// TIA Portal project "EJERCICIO ANALOGIA" (V11)

(* hardware
DEVICE "S7300/ET200 station_1"  SIMATIC 300-Station
   slot 0: "Perfil soporte_0"  Rail  6ES7 390-1***0-0AA0
   slot 2: "PLC_1"  CPU 313C-2 DP  6ES7 313-6CF03-0AB0  V2.6
      slot 0: "Interfaz MPI_1"  MPI
      slot 1: "Interfaz DP_1"  DP
      slot 2: "DI16/DO16_1"  DI16/DO16
      slot 4: "Contaje_1"  Counter
*)

// ===== PLC "PLC_1"  CPU 313C-2 DP =====

VAR_GLOBAL   // PLC tag table "Tabla de variables estándar"
   "Tag_1" AT %E0.0 : Bool;
   "SEÑAL ANALOGICA" AT %MD0 : Real;
   "SALIDA ESCALADO" AT %MD4 : Real;
   "PROPORCIONAL" AT %MD8 : Real;
   "DERIVATIVO" AT %MD12 : Real;
   "INTEGRAL" AT %MD16 : Real;
   "PID" AT %MD20 : Real;
   "BP" AT %MD24 : Real;
   "D" AT %MD28 : Real;
   "I" AT %MD32 : Real;
   "SP" AT %MD36 : Real;
   "valor desescaldo pid" AT %MD40 : Real;
   "porcrntaje apertura valvula" AT %MD44 : Real;
END_VAR

DATA_BLOCK "ESCALADOX_DB"   // DB1
{ S7_Optimized_Access := 'FALSE' }
VERSION : 0.1
// stored: InstanceOfName ESCALADOX
"ESCALADOX"
BEGIN
END_DATA_BLOCK

DATA_BLOCK "DESESCALADO_DB"   // DB2
{ S7_Optimized_Access := 'FALSE' }
VERSION : 0.1
// stored: InstanceOfName DESESCALADO
"DESESCALADO"
BEGIN
END_DATA_BLOCK

DATA_BLOCK "CONTROL PID_DB"   // DB3
{ S7_Optimized_Access := 'FALSE' }
VERSION : 0.1
// stored: InstanceOfName CONTROL PID
"CONTROL PID"
BEGIN
END_DATA_BLOCK

DATA_BLOCK "ESCALADOX_DB_1"   // DB8
{ S7_Optimized_Access := 'FALSE' }
VERSION : 0.1
// stored: InstanceOfName ESCALADOX
"ESCALADOX"
BEGIN
END_DATA_BLOCK

FUNCTION_BLOCK "CONTROL PID"   // FB1, SCL
{ S7_Optimized_Access := 'FALSE' }
VERSION : 0.1
   VAR_INPUT
      SP : Real;
      PV : Real;
      PB : Real;
      D : Real;
      I : Real;
   END_VAR
   VAR_OUTPUT
      "POULT PRO" : Real;
      "POULT DERI" : Real;
      "POULT INTE" : Real;
      "POULT PID PRO" : Real;
   END_VAR
   VAR
      M0 : Bool;
      M1 : Bool;
      T0 : Bool;
      T1 : Bool;
      T2 : Bool;
      T3 : Bool;
      "VISUALIZAR 0" : Time;
      "VISUALIZAR 1" : Time;
      "VISUALIZAR 2" : Time;
      "VISUALIZAR 3" : Time;
      "valor PB" : Real;
      "PB 75 %" : Real;
      "error der inicial" : Real;
      "error int inicial" : Real;
      "error der final" : Real;
      "error int final" : Real;
      ERROR : Real;
      Kp : Real;
      poult : Real;
      Kd : Real;
      "poult der" : Real;
      "diferencia error" : Real;
      Ki : Real;
      "poult int" : Real;
      "incremento error" : Real;
      "aux error integ" : Real;
      "poult pid" : Real;
      Nº100 : Real := 100.0;
      Nº : Real := 0.25;
   END_VAR
BEGIN
END_FUNCTION_BLOCK

FUNCTION_BLOCK "ESCALADOX"   // FB2, SCL
{ S7_Optimized_Access := 'FALSE' }
VERSION : 0.1
   VAR_INPUT
      Y2 : Real;
      Y1 : Real;
      X2 : Real;
      X1 : Real;
      CALCULAR : Bool;
      x : Real;
   END_VAR
   VAR_OUTPUT
      resultado : Real;
   END_VAR
   VAR
      Y : Real;
      "PENDIENTE (m)" : Real;
      "PUNTOCORTE (n)" : Real;
   END_VAR
BEGIN

     #"PENDIENTE (m)" :=  (#Y2 - (#Y1) ) / ( #X2 -#X1   )  ;
     #"PUNTOCORTE (n)" := #Y2  -  #"PENDIENTE (m)" * #X2   ;
     #resultado:= ( #"PENDIENTE (m)" * #x ) + #"PUNTOCORTE (n)";
END_FUNCTION_BLOCK

FUNCTION_BLOCK "DESESCALADO"   // FB3, SCL
{ S7_Optimized_Access := 'FALSE' }
VERSION : 0.1
   VAR_INPUT
      Y2 : Real;
      Y1 : Real;
      X2 : Real;
      X1 : Real;
      "y  valor a desescalar" : Real;
   END_VAR
   VAR_OUTPUT
      "X valor desescalado" : Real;
   END_VAR
   VAR
      "PENDIENTE ( m )" : Real;
      "PUNTO DE CORTE (n )" : Real;
   END_VAR
BEGIN

    #"PENDIENTE ( m )" :=  (#Y2 - (#Y1) ) / ( #X2 -#X1   )  ;
    #"PUNTO DE CORTE (n )" := #Y2  - #"PENDIENTE ( m )" * #X2   ;
    #"X valor desescalado" :=(#"y  valor a desescalar" / #"PENDIENTE ( m )" ) - #"PUNTO DE CORTE (n )" ;
END_FUNCTION_BLOCK

ORGANIZATION_BLOCK "Main"   // OB1, LAD
TITLE = "Main Program Sweep (Cycle)"
{ S7_Optimized_Access := 'FALSE' }
VERSION : 0.1
   VAR_TEMP
      OB1_EV_CLASS : Byte;   // Bits 0-3 = 1 (Coming event), Bits 4-7 = 1 (Event class 1)
      OB1_SCAN_1 : Byte;   // 1 (Cold restart scan 1 of OB 1), 3 (Scan 2-n of OB 1)
      OB1_PRIORITY : Byte;   // Priority of OB Execution
      OB1_OB_NUMBR : Byte;   // 1 (Organization block 1, OB1)
      OB1_RESERVED_1 : Byte;   // Reserved for system
      OB1_RESERVED_2 : Byte;   // Reserved for system
      OB1_PREV_CYCLE : Int;   // Cycle time of previous OB1 scan (milliseconds)
      OB1_MIN_CYCLE : Int;   // Minimum cycle time of OB1 (milliseconds)
      OB1_MAX_CYCLE : Int;   // Maximum cycle time of OB1 (milliseconds)
      OB1_DATE_TIME : Date_And_Time;   // Date and time OB1 started
   END_VAR
BEGIN

REGION Network 1
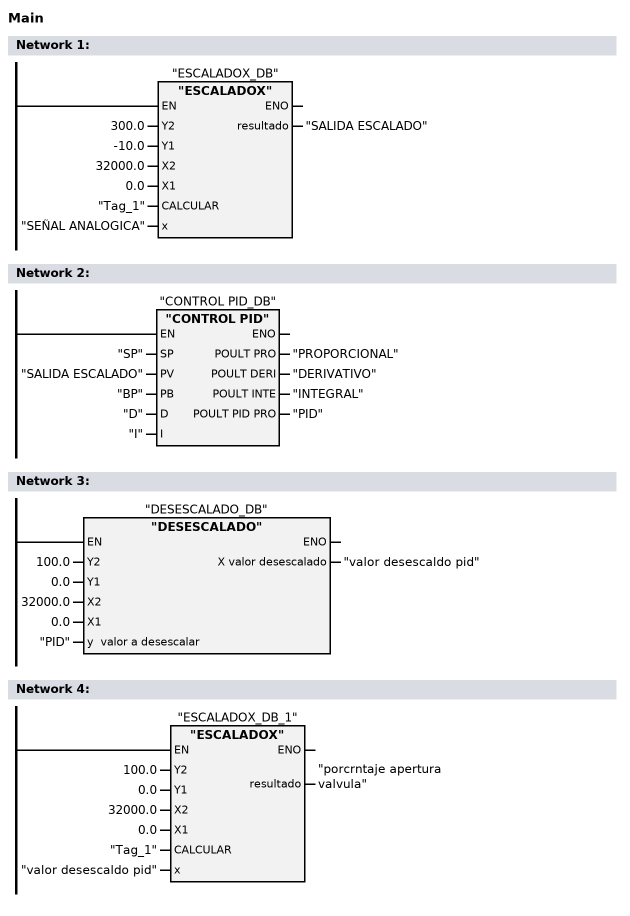
   RUNG wire#powerrail
      "ESCALADOX_DB"(Y2 := 300.0, Y1 := -10.0, X2 := 32000.0, X1 := 0.0, CALCULAR := "Tag_1", x := "SEÑAL ANALOGICA", resultado => "SALIDA ESCALADO")
   END_RUNG
   // the same network as SCL:
   "ESCALADOX_DB"(Y2 := 300.0,   // "ESCALADOX"
                  Y1 := -10.0,
                  X2 := 32000.0,
                  X1 := 0.0,
                  CALCULAR := "Tag_1",
                  x := "SEÑAL ANALOGICA",
                  resultado => "SALIDA ESCALADO");
END_REGION

REGION Network 2
   RUNG wire#powerrail
      "CONTROL PID_DB"(SP := "SP", PV := "SALIDA ESCALADO", PB := "BP", D := "D", I := "I", "POULT PRO" => "PROPORCIONAL", "POULT DERI" => "DERIVATIVO", "POULT INTE" => "INTEGRAL", "POULT PID PRO" => "PID")
   END_RUNG
   // the same network as SCL:
   "CONTROL PID_DB"(SP := "SP",   // "CONTROL PID"
                    PV := "SALIDA ESCALADO",
                    PB := "BP",
                    D := "D",
                    I := "I",
                    "POULT PRO" => "PROPORCIONAL",
                    "POULT DERI" => "DERIVATIVO",
                    "POULT INTE" => "INTEGRAL",
                    "POULT PID PRO" => "PID");
END_REGION

REGION Network 3
   RUNG wire#powerrail
      "DESESCALADO_DB"(Y2 := 100.0, Y1 := 0.0, X2 := 32000.0, X1 := 0.0, "y  valor a desescalar" := "PID", "X valor desescalado" => "valor desescaldo pid")
   END_RUNG
   // the same network as SCL:
   "DESESCALADO_DB"(Y2 := 100.0,   // "DESESCALADO"
                    Y1 := 0.0,
                    X2 := 32000.0,
                    X1 := 0.0,
                    "y  valor a desescalar" := "PID",
                    "X valor desescalado" => "valor desescaldo pid");
END_REGION

REGION Network 4
   RUNG wire#powerrail
      "ESCALADOX_DB_1"(Y2 := 100.0, Y1 := 0.0, X2 := 32000.0, X1 := 0.0, CALCULAR := "Tag_1", x := "valor desescaldo pid", resultado => "porcrntaje apertura valvula")
   END_RUNG
   // the same network as SCL:
   "ESCALADOX_DB_1"(Y2 := 100.0,   // "ESCALADOX"
                    Y1 := 0.0,
                    X2 := 32000.0,
                    X1 := 0.0,
                    CALCULAR := "Tag_1",
                    x := "valor desescaldo pid",
                    resultado => "porcrntaje apertura valvula");
END_REGION
END_ORGANIZATION_BLOCK